INTERFACE PUBLIC I_HoldingCommands

METHOD PUBLIC Abort
END_METHOD

METHOD PUBLIC StateComplete
END_METHOD

METHOD PUBLIC Stop
END_METHOD

END_INTERFACE

(* stored: Version 1.1.0.1, ProductVersion 3.1.4026.6
   Itf I_HoldingCommands: Id {af08fee2-ed8e-0073-1bb5-3408d155c093}
   Method Abort: Id {335d7cb3-9cfd-4dcb-a846-0f0c6849faab}
   Method StateComplete: Id {72815643-eae1-40d6-a359-4dae8ce04b75}
   Method Stop: Id {8b7135c0-a3cd-46c5-83de-1ef3970582a8} *)
